SUBAPPLICATION Dauerfunktion (* Subapplication Type *)
  (* Standard: 61499-2 *)
  (* Version 1.0, 2023-01-29, Franz *)
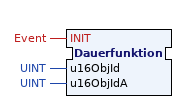
  EVENT_INPUT
    INIT; (* Service Initialization *)
  END_EVENT
  VAR_INPUT
    u16ObjId : UINT;
    u16ObjIdA : UINT;
  END_VAR
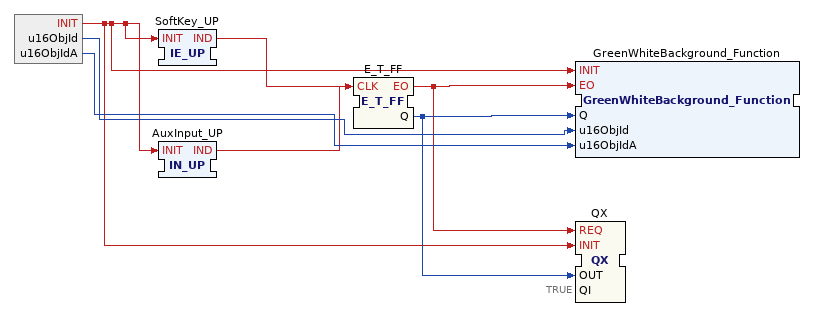
  FBS
    E_T_FF : E_T_FF;
    QX : QX(QI := TRUE);
  END_FBS
  SUBAPPS
    GreenWhiteBackground_Function : GreenWhiteBackground_Function;
    SoftKey_UP : IE_UP;
    AuxInput_UP : IN_UP;
  END_SUBAPPS
  EVENT_CONNECTIONS
    E_T_FF.EO TO QX.REQ;
    INIT TO QX.INIT;
    INIT TO GreenWhiteBackground_Function.INIT;
    E_T_FF.EO TO GreenWhiteBackground_Function.EO;
    INIT TO SoftKey_UP.INIT;
    SoftKey_UP.IND TO E_T_FF.CLK;
    INIT TO AuxInput_UP.INIT;
    AuxInput_UP.IND TO E_T_FF.CLK;
  END_CONNECTIONS
  DATA_CONNECTIONS
    E_T_FF.Q TO QX.OUT;
    E_T_FF.Q TO GreenWhiteBackground_Function.Q;
    u16ObjId TO GreenWhiteBackground_Function.u16ObjId;
    u16ObjIdA TO GreenWhiteBackground_Function.u16ObjIdA;
  END_CONNECTIONS
END_SUBAPPLICATION
